TYPE TcoDatamanIO_v_5_x_x :
STRUCT
	PnIoBoxState AT %I*	:	UINT;
	PnIoBoxDiag AT %I*	:	UINT;
	PnIoBoxCtrl AT %Q*	:	UINT;
	AcquisitionControl	:	TcoDatamanAcquisitionControl_v_5_x_x;
	AcquisitionStatus	:	TcoDatamanAcquisitionStatus_v_5_x_x;
	ResultsControl		:	TcoDatamanResultsControl_v_5_x_x;
	ResultsStatus		:	TcoDatamanResultsStatus_v_5_x_x;
	SoftEventControl	:	TcoDatamanSoftEventControl_v_5_x_x;
	UserData			:	TcoDatamanUserData_v_5_x_x;
	ResultData			:	TcoDatamanResultData_v_5_x_x;
END_STRUCT
END_TYPE

(* stored: Version 1.1.0.1, ProductVersion 3.1.4024.11
   DUT TcoDatamanIO_v_5_x_x: Id {15e8d456-5b4f-4523-9246-2822fb48f181} *)
